% RSLogix 500 project LAB 2 AUTO new.RSS, saved by version 8.40.00.08 %
PROJECT "UNTITLED"    % processor: type code 33 %

PROGRAM FILES
  LAD 2   38 rungs

DATA FILES
  O0 OUTPUT  68 elements
  I1 INPUT  68 elements
  S2 STATUS  164 elements
  B3 BINARY  2 elements
  T4 TIMER  34 elements
  C5 COUNTER  35 elements
  R6 CONTROL  1 elements
  N7 INTEGER  1 elements
  F8 FLOAT  1 elements

LADDER 2
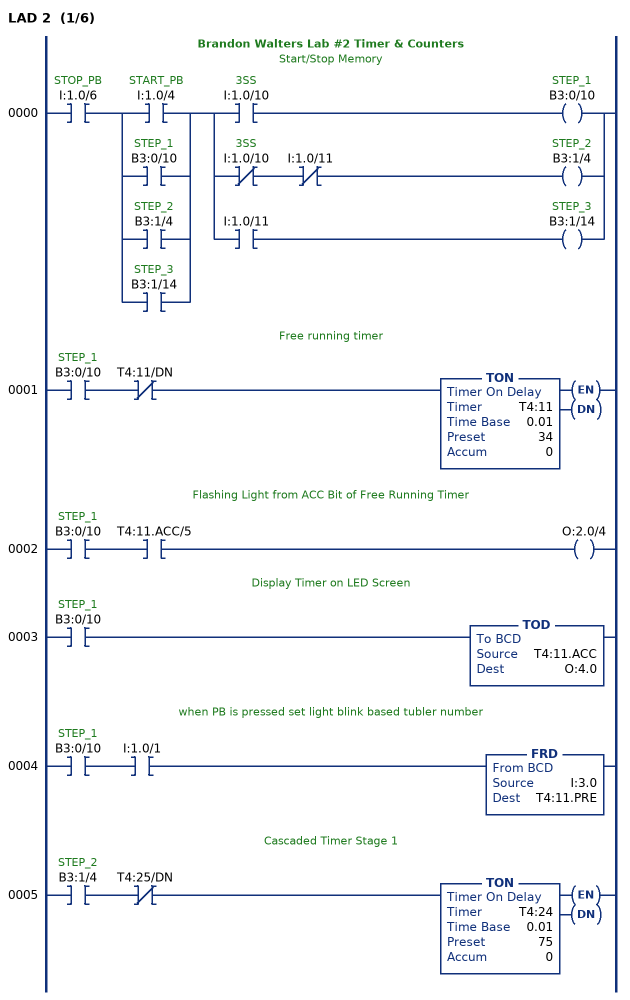
% Rung: 0 %
% TITLE: Brandon Walters Lab #2 Timer & Counters %
% Start/Stop Memory %
SOR XIC I:1.0/6 BST XIC I:1.0/4 NXB XIC B3:0/10 NXB XIC B3:1/4 NXB XIC B3:1/14 BND BST XIC I:1.0/10 OTE B3:0/10 NXB XIO I:1.0/10 XIO I:1.0/11 OTE B3:1/4 NXB XIC I:1.0/11 OTE B3:1/14 BND EOR
%   I:1.0/6  STOP_PB %
%   I:1.0/4  START_PB %
%   B3:0/10  STEP_1 %
%   B3:1/4  STEP_2 %
%   B3:1/14  STEP_3 %
%   I:1.0/10  3SS %
% Rung: 1 %
% Free running timer %
SOR XIC B3:0/10 XIO T4:11/DN TON T4:11 0.01 34 0 EOR
%   B3:0/10  STEP_1 %
% Rung: 2 %
% Flashing Light from ACC Bit of Free Running Timer %
SOR XIC B3:0/10 XIC T4:11.ACC/5 OTE O:2.0/4 EOR
%   B3:0/10  STEP_1 %
% Rung: 3 %
% Display Timer on LED Screen %
SOR XIC B3:0/10 TOD T4:11.ACC O:4.0 EOR
%   B3:0/10  STEP_1 %
% Rung: 4 %
% when PB is pressed set light blink based tubler number %
SOR XIC B3:0/10 XIC I:1.0/1 FRD I:3.0 T4:11.PRE EOR
%   B3:0/10  STEP_1 %
% Rung: 5 %
% Cascaded Timer Stage 1 %
SOR XIC B3:1/4 XIO T4:25/DN TON T4:24 0.01 75 0 EOR
%   B3:1/4  STEP_2 %

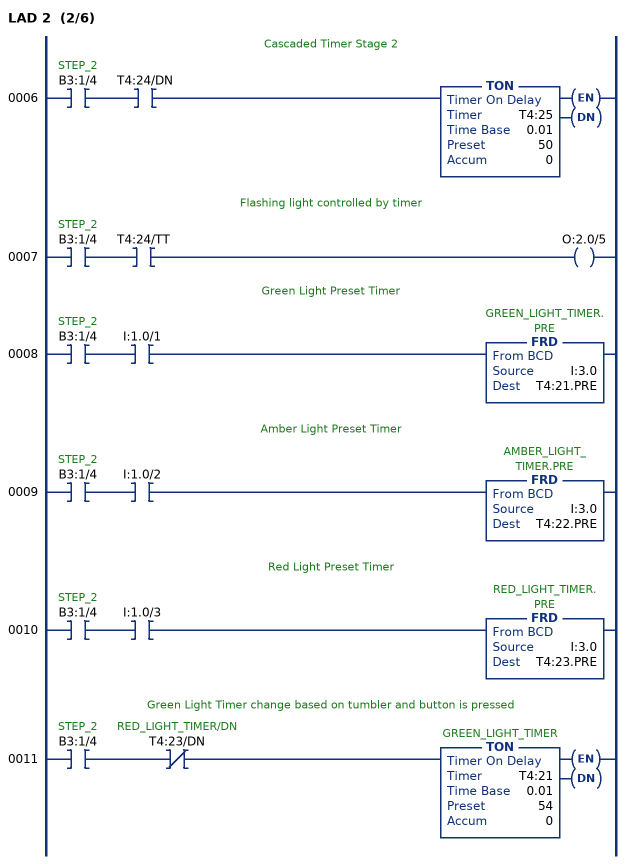
% Rung: 6 %
% Cascaded Timer Stage 2 %
SOR XIC B3:1/4 XIC T4:24/DN TON T4:25 0.01 50 0 EOR
%   B3:1/4  STEP_2 %
% Rung: 7 %
% Flashing light controlled by timer %
SOR XIC B3:1/4 XIC T4:24/TT OTE O:2.0/5 EOR
%   B3:1/4  STEP_2 %
% Rung: 8 %
% Green Light Preset Timer %
SOR XIC B3:1/4 XIC I:1.0/1 FRD I:3.0 T4:21.PRE EOR
%   B3:1/4  STEP_2 %
%   T4:21  GREEN_LIGHT_TIMER %
% Rung: 9 %
% Amber Light Preset Timer %
SOR XIC B3:1/4 XIC I:1.0/2 FRD I:3.0 T4:22.PRE EOR
%   B3:1/4  STEP_2 %
%   T4:22  AMBER_LIGHT_TIMER %
% Rung: 10 %
% Red Light Preset Timer %
SOR XIC B3:1/4 XIC I:1.0/3 FRD I:3.0 T4:23.PRE EOR
%   B3:1/4  STEP_2 %
%   T4:23  RED_LIGHT_TIMER %
% Rung: 11 %
% Green Light Timer change based on tumbler and button is pressed %
SOR XIC B3:1/4 XIO T4:23/DN TON T4:21 0.01 54 0 EOR
%   B3:1/4  STEP_2 %
%   T4:23  RED_LIGHT_TIMER %
%   T4:21  GREEN_LIGHT_TIMER %

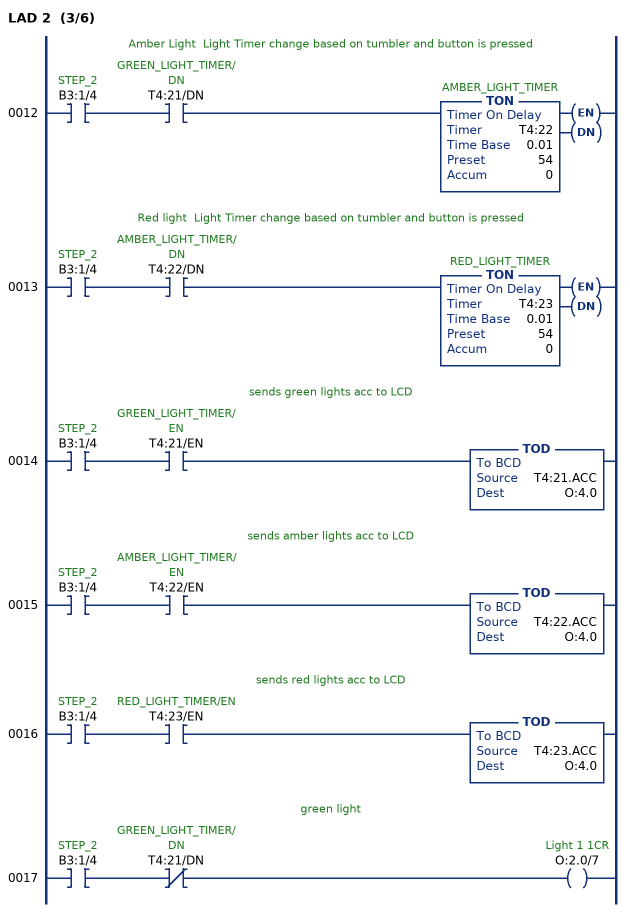
% Rung: 12 %
% Amber Light  Light Timer change based on tumbler and button is pressed %
SOR XIC B3:1/4 XIC T4:21/DN TON T4:22 0.01 54 0 EOR
%   B3:1/4  STEP_2 %
%   T4:21  GREEN_LIGHT_TIMER %
%   T4:22  AMBER_LIGHT_TIMER %
% Rung: 13 %
% Red light  Light Timer change based on tumbler and button is pressed %
SOR XIC B3:1/4 XIC T4:22/DN TON T4:23 0.01 54 0 EOR
%   B3:1/4  STEP_2 %
%   T4:22  AMBER_LIGHT_TIMER %
%   XIC T4:22/DN  "Amber Light Done Red Starts" %
%   T4:23  RED_LIGHT_TIMER %
% Rung: 14 %
% sends green lights acc to LCD %
SOR XIC B3:1/4 XIC T4:21/EN TOD T4:21.ACC O:4.0 EOR
%   B3:1/4  STEP_2 %
%   T4:21  GREEN_LIGHT_TIMER %
% Rung: 15 %
% sends amber lights acc to LCD %
SOR XIC B3:1/4 XIC T4:22/EN TOD T4:22.ACC O:4.0 EOR
%   B3:1/4  STEP_2 %
%   T4:22  AMBER_LIGHT_TIMER %
% Rung: 16 %
% sends red lights acc to LCD %
SOR XIC B3:1/4 XIC T4:23/EN TOD T4:23.ACC O:4.0 EOR
%   B3:1/4  STEP_2 %
%   T4:23  RED_LIGHT_TIMER %
% Rung: 17 %
% green light %
SOR XIC B3:1/4 XIO T4:21/DN OTE O:2.0/7 EOR
%   B3:1/4  STEP_2 %
%   T4:21  GREEN_LIGHT_TIMER %
%   O:2.0/7  1CR  "Light 1" %

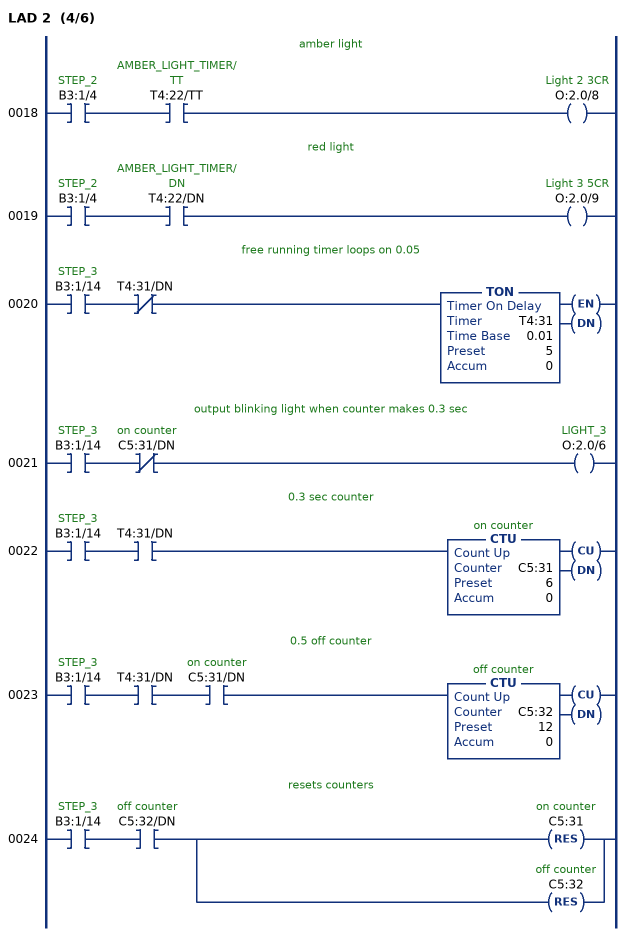
% Rung: 18 %
% amber light %
SOR XIC B3:1/4 XIC T4:22/TT OTE O:2.0/8 EOR
%   B3:1/4  STEP_2 %
%   T4:22  AMBER_LIGHT_TIMER %
%   O:2.0/8  3CR  "Light 2" %
% Rung: 19 %
% red light %
SOR XIC B3:1/4 XIC T4:22/DN OTE O:2.0/9 EOR
%   B3:1/4  STEP_2 %
%   T4:22  AMBER_LIGHT_TIMER %
%   XIC T4:22/DN  "Amber Light Done Red Starts" %
%   O:2.0/9  5CR  "Light 3" %
% Rung: 20 %
% free running timer loops on 0.05 %
SOR XIC B3:1/14 XIO T4:31/DN TON T4:31 0.01 5 0 EOR
%   B3:1/14  STEP_3 %
% Rung: 21 %
% output blinking light when counter makes 0.3 sec %
SOR XIC B3:1/14 XIO C5:31/DN OTE O:2.0/6 EOR
%   B3:1/14  STEP_3 %
%   C5:31  "on counter" %
%   O:2.0/6  LIGHT_3 %
% Rung: 22 %
% 0.3 sec counter %
SOR XIC B3:1/14 XIC T4:31/DN CTU C5:31 6 0 EOR
%   B3:1/14  STEP_3 %
%   C5:31  "on counter" %
% Rung: 23 %
% 0.5 off counter %
SOR XIC B3:1/14 XIC T4:31/DN XIC C5:31/DN CTU C5:32 12 0 EOR
%   B3:1/14  STEP_3 %
%   C5:31  "on counter" %
%   C5:32  "off counter" %
% Rung: 24 %
% resets counters %
SOR XIC B3:1/14 XIC C5:32/DN BST RES C5:31 NXB RES C5:32 BND EOR
%   B3:1/14  STEP_3 %
%   C5:32  "off counter" %
%   C5:31  "on counter" %

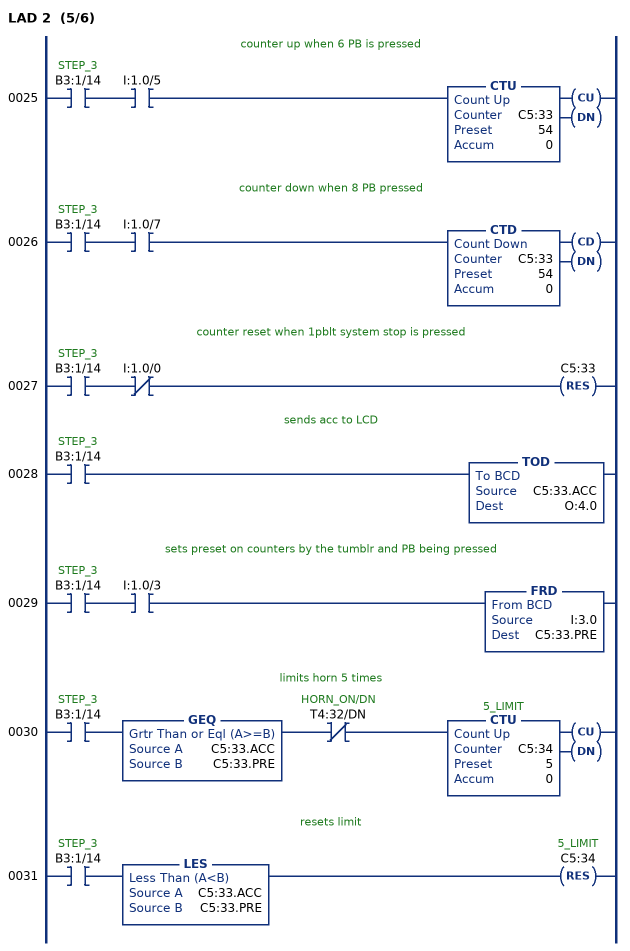
% Rung: 25 %
% counter up when 6 PB is pressed %
SOR XIC B3:1/14 XIC I:1.0/5 CTU C5:33 54 0 EOR
%   B3:1/14  STEP_3 %
% Rung: 26 %
% counter down when 8 PB pressed %
SOR XIC B3:1/14 XIC I:1.0/7 CTD C5:33 54 0 EOR
%   B3:1/14  STEP_3 %
% Rung: 27 %
% counter reset when 1pblt system stop is pressed %
SOR XIC B3:1/14 XIO I:1.0/0 RES C5:33 EOR
%   B3:1/14  STEP_3 %
% Rung: 28 %
% sends acc to LCD %
SOR XIC B3:1/14 TOD C5:33.ACC O:4.0 EOR
%   B3:1/14  STEP_3 %
% Rung: 29 %
% sets preset on counters by the tumblr and PB being pressed %
SOR XIC B3:1/14 XIC I:1.0/3 FRD I:3.0 C5:33.PRE EOR
%   B3:1/14  STEP_3 %
% Rung: 30 %
% limits horn 5 times %
SOR XIC B3:1/14 GEQ C5:33.ACC C5:33.PRE XIO T4:32/DN CTU C5:34 5 0 EOR
%   B3:1/14  STEP_3 %
%   T4:32  HORN_ON %
%   C5:34  5_LIMIT %
% Rung: 31 %
% resets limit %
SOR XIC B3:1/14 LES C5:33.ACC C5:33.PRE RES C5:34 EOR
%   B3:1/14  STEP_3 %
%   C5:34  5_LIMIT %

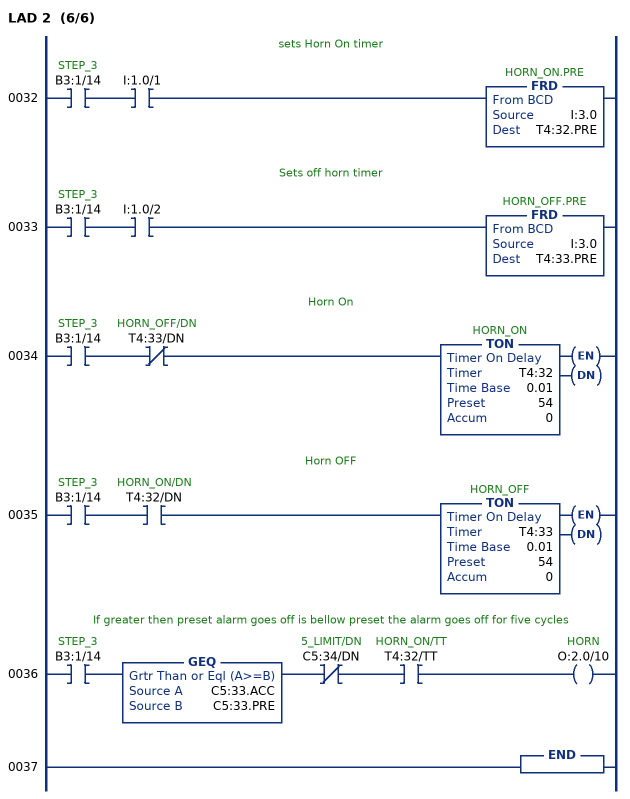
% Rung: 32 %
% sets Horn On timer %
SOR XIC B3:1/14 XIC I:1.0/1 FRD I:3.0 T4:32.PRE EOR
%   B3:1/14  STEP_3 %
%   T4:32  HORN_ON %
% Rung: 33 %
% Sets off horn timer %
SOR XIC B3:1/14 XIC I:1.0/2 FRD I:3.0 T4:33.PRE EOR
%   B3:1/14  STEP_3 %
%   T4:33  HORN_OFF %
% Rung: 34 %
% Horn On %
SOR XIC B3:1/14 XIO T4:33/DN TON T4:32 0.01 54 0 EOR
%   B3:1/14  STEP_3 %
%   T4:33  HORN_OFF %
%   T4:32  HORN_ON %
% Rung: 35 %
% Horn OFF %
SOR XIC B3:1/14 XIC T4:32/DN TON T4:33 0.01 54 0 EOR
%   B3:1/14  STEP_3 %
%   T4:32  HORN_ON %
%   T4:33  HORN_OFF %
% Rung: 36 %
% If greater then preset alarm goes off is bellow preset the alarm goes off for five cycles %
SOR XIC B3:1/14 GEQ C5:33.ACC C5:33.PRE XIO C5:34/DN XIC T4:32/TT OTE O:2.0/10 EOR
%   B3:1/14  STEP_3 %
%   C5:34  5_LIMIT %
%   T4:32  HORN_ON %
%   O:2.0/10  HORN %
% Rung: 37 %
SOR END EOR

OTHER DOCUMENTED ADDRESSES
  B3:0/2  2CR
  B3:0/4  4CR
  B3:0/6  6CR
  B3:0/7  7CR  "Reset"
  I:1.0/8  1SS
  I:1.0/9  2SS
  O:2.0/1  2PBLT
  O:2.0/2  3PBLT
  O:2.0/3  4PBLT

DATA TABLE (non-zero values as saved)
DATA T4
% .PRE .ACC %
% T4:11 % 34 0
% T4:21 % 54 0
% T4:22 % 54 0
% T4:23 % 54 0
% T4:24 % 75 0
% T4:25 % 50 0
% T4:31 % 5 0
% T4:32 % 54 0
% T4:33 % 54 0
DATA C5
% .PRE .ACC %
% C5:31 % 6 0
% C5:32 % 12 0
% C5:33 % 54 0
% C5:34 % 5 0
